// TIA Portal V20 export
DATA_BLOCK "Sen"   // DB324
{ S7_Optimized_Access := 'TRUE' }
// stored: AutoNumber false, IsRetainMemResEnabled true, MemoryReserve 500, RetainMemoryReserve 500
   VAR RETAIN
      "1BTR2+SGV" : "TypeSensor";   // light barrier in scannerhousing visual measurement
      "1BTR2+SGX" : "TypeSensor";   // light barrier in scannerhousing x-ray measurement
      "8S1.T" : "TypeSensor";   // adjustment top limit switch innermost position
      "8S2.T" : "TypeSensor";   // adjustment top limit switch outermost position
      "8S1.L" : "TypeSensor";   // adjustment left limit switch innermost position
      "8S2.L" : "TypeSensor";   // adjustment left limit switch outermost position
      "8S1.R" : "TypeSensor";   // adjustment right limit switch innermost position
      "8S2.R" : "TypeSensor";   // adjustment right limit switch outermost position
      "8S1.B" : "TypeSensor";   // adjustment scanner limit switch left position
      "8S2.B" : "TypeSensor";   // adjustment scanner limit switch right position
      "8B1" : "TypeSensor";   // light barrier measuring distance top
      "8B2" : "TypeSensor";   // light barrier measuring distance left
      "8B3" : "TypeSensor";   // light barrier measuring distance right
   END_VAR
BEGIN
   "1BTR2+SGV".description := WSTRING#'Sensor Aufgabförderer 1 Ende belegt - Zubringung';
   "1BTR2+SGX".description := WSTRING#'Sensor Aufgabförderer 2 Ende belegt - Zubringung';
   "8S1.T".description := WSTRING#'Sensor Aufgabförderer 2 Ende belegt - Zubringung';
   "8S2.T".description := WSTRING#'Sensor Aufgabförderer 2 Ende belegt - Zubringung';
   "8S1.L".description := WSTRING#'Sensor Aufgabförderer 2 Ende belegt - Zubringung';
   "8S2.L".description := WSTRING#'Sensor Aufgabförderer 2 Ende belegt - Zubringung';
   "8S1.R".description := WSTRING#'Sensor Aufgabförderer 2 Ende belegt - Zubringung';
   "8S2.R".description := WSTRING#'Sensor Aufgabförderer 2 Ende belegt - Zubringung';
   "8S1.B".description := WSTRING#'Sensor Aufgabförderer 2 Ende belegt - Zubringung';
   "8S2.B".description := WSTRING#'Sensor Aufgabförderer 2 Ende belegt - Zubringung';
END_DATA_BLOCK
